{attribute addProperty BoxType "EL1252-0000-0018"}
{attribute addProperty Id "Status1AT %I*USINT81174Status2AT %I*USINT81175LatchPos1AT %I*ULINT648176LatchNeg1AT %I*ULINT648184LatchPos2AT %I*ULINT648192LatchNeg2AT %I*ULINT648200"}
{attribute addProperty CRC "290304593"}
{attribute addProperty SizeInBites "272"}
{attribute addProperty SizeInBytes "34"}
TYPE Latch_114DB251 :
STRUCT
	{attribute addProperty Name "Status1"}
	Status1 AT %I* : USINT;
	{attribute addProperty Name "Status2"}
	Status2 AT %I* : USINT;
	{attribute addProperty Name "LatchPos1"}
	LatchPos1 AT %I* : ULINT;
	{attribute addProperty Name "LatchNeg1"}
	LatchNeg1 AT %I* : ULINT;
	{attribute addProperty Name "LatchPos2"}
	LatchPos2 AT %I* : ULINT;
	{attribute addProperty Name "LatchNeg2"}
	LatchNeg2 AT %I* : ULINT;
END_STRUCT
END_TYPE

(* stored: Version 1.2.0.0, ProductVersion 3.1.4024.9
   DUT Latch_114DB251: Id {63bcaad6-0dd4-4b1b-a129-bbe5c5d340c5} *)
